FUNCTION_BLOCK FB_Greifer EXTENDS GrundstrukturObjekt
VAR_INPUT
END_VAR
VAR_OUTPUT
END_VAR
VAR
END_VAR

END_FUNCTION_BLOCK

(* stored: Version 1.1.0.1
   POU FB_Greifer: Id {29489103-a9cc-4ccd-8b54-c54ca0ae9cd0}, SpecialFunc None *)
